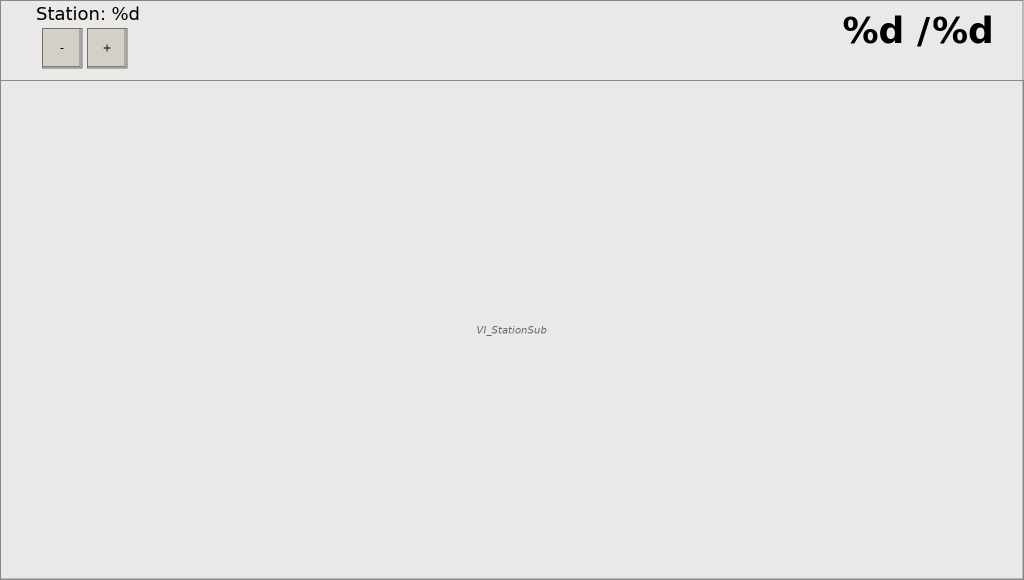
VISUALIZATION VI_Station  // 1024x580
    Frame (0,80 1024x500)
        shows VI_StationSub()
    Rectangle (929,5 77x51), "%d", text variable: GVL_XPlanarVisuDiag.nMaxStationToDisplay
    Rectangle (830,5 103x51), "%d /", text variable: GVL_XPlanarVisuDiag.nStationIdToDisplay
    Button (87,28 40x40), "+", invisible if: GVL_StationVisu.bStationNextInvisible
        tap GVL_XPlanarVisuDiag.bStationNext p1329445385=TRUE
    Button (42,28 40x40), "-", invisible if: GVL_XPlanarVisuDiag.bSationPreviousInvisible
        tap GVL_XPlanarVisuDiag.bStationPrevious
    Rectangle (34,2 108x24), "Station: %d", text variable: GVL_XPlanarVisuDiag.nStationIdToDisplay
END_VISUALIZATION

(* stored: Version 1.1.0.1, ProductVersion 3.1.4024.9
   Visu VI_Station: Id {e973bd10-3f81-41f0-972c-fd9105037b3a} *)
